// Implicitly generated code : DO NOT EDIT
FUNCTION CheckDivReal : REAL
VAR_INPUT
	divisor:REAL;
END_VAR

// Implicitly generated code : Only an Implementation suggestion
{noflow}
IF divisor = 0 THEN
	CheckDivReal:=1;
	G_Diag.uiCheckDivReal:=G_Diag.uiCheckDivReal+1;
ELSE
	CheckDivReal:=divisor;
END_IF;
{flow}

END_FUNCTION

(* stored: Version 1.1.0.1, ProductVersion 3.1.4024.4
   POU CheckDivReal: Id {4a4e550e-9e6c-4c92-a948-5ed0dd3c97b0}, SpecialFunc CheckDivReal32 *)
